FUNCTION_BLOCK TEST_SH2 (* Test DWORD, LWORD shift functions *)
  (* Standard: 61499-1 *)
  (* Version 0.1, 2007-11-11, JHC, Holobloc Inc, Deleted import. *)
  (* Version 0.0, 2006-09-06, JHC, Holobloc Inc *)
  (* Compiler header: package fb.rt.test; *)
  (* Compiler classdef: SimpleFB *)
  (* Compiler Java Sun JDK 1.6.0 *)
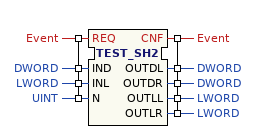
  EVENT_INPUT
    REQ WITH IND, INL, N; (* Normal Execution Request *)
  END_EVENT
  EVENT_OUTPUT
    CNF WITH OUTDL, OUTDR, OUTLL, OUTLR; (* Execution Confirmation *)
  END_EVENT
  VAR_INPUT
    IND : DWORD;
    INL : LWORD;
    N : UINT;
  END_VAR
  VAR_OUTPUT
    OUTDL : DWORD;
    OUTDR : DWORD;
    OUTLL : LWORD;
    OUTLR : LWORD;
  END_VAR
  ALGORITHM REQ IN FBD: (* Normally executed algorithm *)
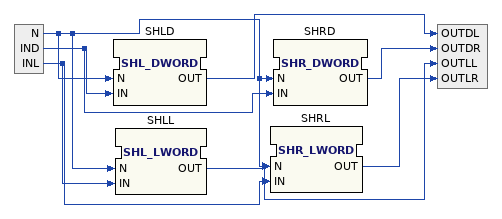
    FBS
      SHLD : SHL_DWORD;
      SHRD : SHR_DWORD;
      SHLL : SHL_LWORD;
      SHRL : SHR_LWORD;
    END_FBS
    DATA_CONNECTIONS
      N TO SHLD.N;
      N TO SHRD.N;
      N TO SHLL.N;
      N TO SHRL.N;
      IND TO SHLD.IN;
      SHLD.OUT TO OUTDL;
      IND TO SHRD.IN;
      SHRD.OUT TO OUTDR;
      INL TO SHLL.IN;
      SHLL.OUT TO OUTLL;
      INL TO SHRL.IN;
      SHRL.OUT TO OUTLR;
    END_CONNECTIONS
  END_ALGORITHM
END_FUNCTION_BLOCK
